PROGRAM MAIN
VAR
END_VAR

END_PROGRAM

(* stored: Version 1.1.0.1
   POU MAIN: Id {598522ef-285b-48b1-8c04-34d19fe25b62} *)
